PROGRAM mainBranch
VAR
END_VAR

END_PROGRAM

(* stored: Version 1.1.0.1, ProductVersion 3.1.4024.12
   POU mainBranch: Id {0d212e3f-3bd6-0024-34c7-95813e41232f}, SpecialFunc None *)
